PROGRAM MAIN
VAR
	fbCircle : FB_Circle;
	fbGreenCircle : FB_GreenShapeDecorator(fbCircle);
	fbRoundDotBorderGreenCircle : FB_BorderDashTypeDecorator(fbGreenCircle,E_BorderDashType.RoundDot);
	
	fbSquare : FB_Square;
	fbGreenSquare : FB_GreenShapeDecorator(fbSquare);
	fbDashBorderGreenSquare : FB_BorderDashTypeDecorator(fbGreenSquare,E_BorderDashType.Dash);
	
	bDemoStart: BOOL;
END_VAR


IF bDemoStart THEN
	
	bDemoStart := FALSE;
	
	fbRoundDotBorderGreenCircle.M_Draw();

	fbDashBorderGreenSquare.M_Draw();

END_IF

END_PROGRAM

(* stored: Version 1.1.0.1, ProductVersion 3.1.4024.12
   POU MAIN: Id {6fe1dd67-29d5-4d6b-b525-e0ff86671bb2}, SpecialFunc None *)
